// TIA Portal V20 export
DATA_BLOCK "RealDbName"   // DB7
   VAR
      LockedFlag { ExternalWritable := 'False'} : Bool;
   END_VAR
BEGIN
END_DATA_BLOCK
